(* PLC project motor_2dir_2speed, Dassault Systèmes ControlBuild 2024x *)
(* stored: creationDateTime 2023-10-03T11:13:09-01:00 *)

(* This module simulates the behaviour of a motor with 2 directions et 2 speeds and its electrical control logic. *)
FUNCTION_BLOCK equipment_library.motor_2dir_2speed
  VAR_INPUT
    voltage380 : BOOL := true;
    cmdSupply : BOOL := true;
    sensorSupply : BOOL := true;
  END_VAR
  VAR_INPUT
    forward : BOOL := false;
    backward : BOOL := false;
    highSpeed : BOOL := false;
    lowSpeed : BOOL := false;
  END_VAR
  VAR_OUTPUT
    forwardFB : BOOL := false;
    backwardFB : BOOL := false;
    highSpeedFB : BOOL := false;
    lowSpeedFB : BOOL := false;
    thermal : BOOL := false;
  END_VAR
  VAR_OUTPUT
    speedVal : REAL := 0.0;
    speedPercent : REAL := 0.0;
  END_VAR
  VAR
    increment : REAL := 0.0;
    memoFwd : BOOL := false;
    memoBwd : BOOL := false;
    memoHighSpeed : BOOL := false;
    memoLowSpeed : BOOL := false;
    FwdHsState : BOOL := false;
    FwdLsState : BOOL := false;
    BwdHsState : BOOL := false;
    BwdLsState : BOOL := false;
    wantedSpeed : REAL := 0.0;
  END_VAR
  VAR CONSTANT
    nominalTime : REAL := 0.5;
    thermalLogic : BOOL := false;
    fwdFbLogic : BOOL := true;
    bwdFbLogic : BOOL := true;
    highSpeedFbLogic : BOOL := true;
    lowSpeedFbLogic : BOOL := true;
    nominalLowSpeed : REAL := 2500.0;
    nominalHighSpeed : REAL := 5000.0;
  END_VAR
  VAR
    d_locking : BOOL := false;
    v_d_locking : REAL := 0.5;
    d_electrical : BOOL := false;
    v_d_electrical : BOOL := false;
    d_forwardFB : BOOL := false;
    v_d_forwardFB : BOOL := false;
    d_highSpeedFB : BOOL := false;
    v_d_highSpeedFB : BOOL := false;
    d_lowSpeedFB : BOOL := false;
    v_d_lowSpeedFB : BOOL := false;
    d_backwardFB : BOOL := false;
    v_d_backwardFB : BOOL := false;
  END_VAR


ACTION C_source_code:
/* ----------------------------------------------------------------	*/
/* Type : Model of Operative Behaviour					*/
/* Category :  Associations - motors					*/
/* Author : Dassault Systemes						*/
/* Update date : June 2010							*/
/* ----------------------------------------------------------------	*/
/* This module simulates a motor with 2 directions and 2 speeds	*/
/* and its electrical control logic.					*/
/* ----------------------------------------------------------------	*/


/* ----------------------------------------------------------------	*/
/* Management of orders from Control Part					*/
/*	if there is no power supply for command 				*/
/*     	the contactors don't understand the control order	*/
/*	The contactors cannot be active in the same time		*/
/*	 	(mechanical security).					*/
/* ----------------------------------------------------------------	*/
if (forward && !memoBwd && cmdSupply) memoFwd = 1;
if (!forward || !cmdSupply || d_electrical) memoFwd = 0;
if (!memoFwd && backward && cmdSupply) memoBwd = 1;
if (!backward || !cmdSupply || d_electrical) memoBwd = 0;

if (!memoHighSpeed && lowSpeed && cmdSupply) memoLowSpeed = 1;
if (!lowSpeed || !cmdSupply || d_electrical) memoLowSpeed = 0;
if (highSpeed && !memoLowSpeed && cmdSupply) memoHighSpeed = 1;
if (!highSpeed || !cmdSupply || d_electrical) memoHighSpeed = 0;

/* ----------------------------------------------------------------	*/
/* Calculation of the on-state of contactor				*/
/* ----------------------------------------------------------------	*/
FwdHsState = memoFwd & memoHighSpeed & voltage380;
FwdLsState = memoFwd & memoLowSpeed & voltage380;
BwdHsState = memoBwd & memoHighSpeed & voltage380;
BwdLsState = memoBwd & memoLowSpeed & voltage380;


/* ----------------------------------------------------------------	*/
/* Management of the speed ramp						*/
/* ----------------------------------------------------------------	*/
if (d_locking)  speedVal = v_d_locking;
else {
	/* compute the wanted speed	*/
	if (FwdHsState) {
		wantedSpeed = nominalHighSpeed;
		if (nominalTime > 0.0)
			increment=(nominalHighSpeed/nominalTime)*(CLOCK_PERIOD/1000000.0);
	}
	else if (FwdLsState) {
		wantedSpeed = nominalLowSpeed;
		if (nominalTime > 0.0)
			increment=(nominalLowSpeed/nominalTime)*(CLOCK_PERIOD/1000000.0);
	}
	if (BwdHsState) {
		wantedSpeed = nominalHighSpeed * -1.0;
		increment=(nominalHighSpeed/nominalTime)*(CLOCK_PERIOD/1000000.0);
	}
	else if (BwdLsState) {
		wantedSpeed = nominalLowSpeed * -1.0;
		increment=(nominalLowSpeed/nominalTime)*(CLOCK_PERIOD/1000000.0);
	}
	 if (! FwdHsState && ! FwdLsState && ! BwdHsState && ! BwdLsState) wantedSpeed = 0.0;


	/* Compute the speed ramp	*/
	if ( speedVal < wantedSpeed) {
		speedVal += increment;
		if ( speedVal > wantedSpeed) speedVal = wantedSpeed;
	}
	if ( speedVal > wantedSpeed) {
		speedVal -= increment;
		if (speedVal < wantedSpeed) speedVal = wantedSpeed;
	}
}

/* ----------------------------------------------------------------	*/
/* Compute the percentage between the current and nominal speed	*/
/* ----------------------------------------------------------------	*/
if (nominalHighSpeed != 0.0)
	speedPercent = ((speedVal/nominalHighSpeed)*100);

/* ----------------------------------------------------------------	*/
/* Management of the thermal feedback					*/
/* ----------------------------------------------------------------	*/
if (d_electrical) thermal=v_d_electrical;
else
	thermal= ! thermalLogic && sensorSupply;

/* ----------------------------------------------------------------	*/
/* Management of feedback to Control Part					*/
/*     if a fault is required, the contactor feed-back 		*/
/*		 takes a preset state.					*/
/*	if there is no power supply for sensors 				*/
/*         contactor feed-back returns nothing				*/
/*     else contactor feed-back returns the contactor state combined	*/
/*	    with wiring logic.						*/
/* ----------------------------------------------------------------	*/
if (d_forwardFB) forwardFB = v_d_forwardFB;
else
	forwardFB=(memoFwd ^ ! fwdFbLogic) && sensorSupply;

if (d_backwardFB) backwardFB = v_d_backwardFB;
else
	backwardFB = (memoBwd ^ ! bwdFbLogic) && sensorSupply;

if (d_highSpeedFB) highSpeedFB = v_d_highSpeedFB;
else
	highSpeedFB = (memoHighSpeed ^ ! highSpeedFbLogic) && sensorSupply;

if (d_lowSpeedFB) lowSpeedFB = v_d_lowSpeedFB;
else
	lowSpeedFB = (memoLowSpeed ^ ! lowSpeedFbLogic) && sensorSupply;
END_ACTION
END_FUNCTION_BLOCK
